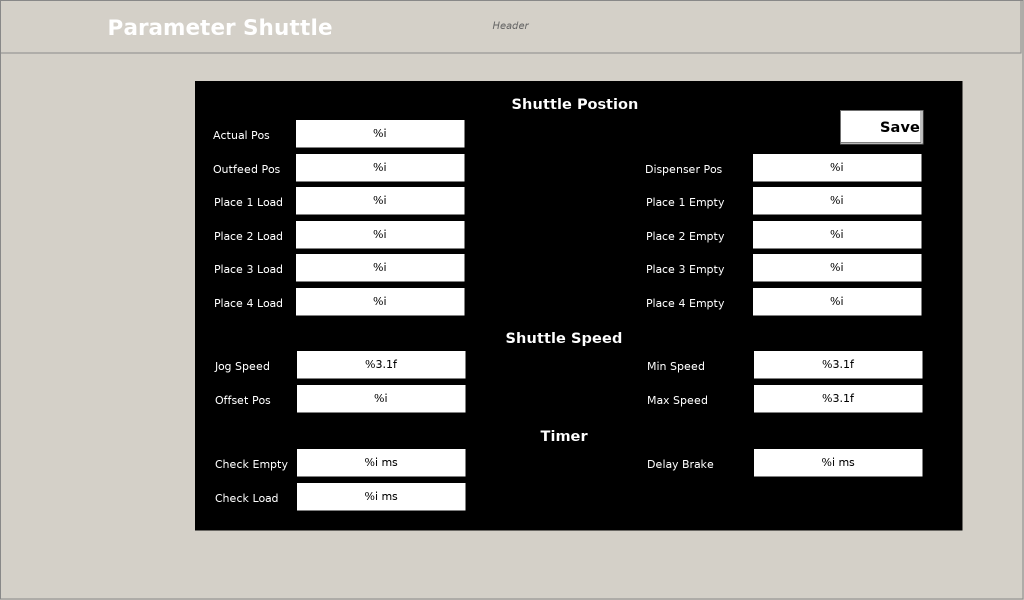
VISUALIZATION MShuttle  // 1024x600
    Frame (0,-2 1021x55)
        shows Header()
    Label (95,15 250x25), "Parameter Shuttle"
    RoundedRectangle (195,81 767x449)
    Label (223,84 704x40), "Shuttle Postion"
    Label (210,118 78x35), "Actual Pos"
    RoundedRectangle (295,119 170x29), "%i", text variable: InputOutput_GVL.ShuttlePosition
    Button (840,110 83x34), "Save", image: VisuSymbols.Symbols.Save
        tap InputOutput_GVL.TestMode[100]
    Label (210,152 78x35), "Outfeed Pos"
    RoundedRectangle (295,153 170x29), "%i", text variable: HMI_GVL.stShuttleSequence[0].PositionLoaded
        OnMouseClick: write the text variable via Default
    Label (642,152 102x35), "Dispenser Pos"
    RoundedRectangle (752,153 170x29), "%i", text variable: HMI_GVL.stShuttleSequence[0].PositionEmpty
        OnMouseClick: write the text variable via Default
    Label (211,185 78x35), "Place 1 Load"
    RoundedRectangle (295,186 170x29), "%i", text variable: HMI_GVL.stShuttleSequence[1].PositionLoaded
        OnMouseClick: write the text variable via Default
    Label (643,185 102x35), "Place 1 Empty"
    RoundedRectangle (752,186 170x29), "%i", text variable: HMI_GVL.stShuttleSequence[1].PositionEmpty
        OnMouseClick: write the text variable via Default
    Label (211,219 78x35), "Place 2 Load"
    RoundedRectangle (295,220 170x29), "%i", text variable: HMI_GVL.stShuttleSequence[2].PositionLoaded
        OnMouseClick: write the text variable via Default
    Label (643,219 102x35), "Place 2 Empty"
    RoundedRectangle (752,220 170x29), "%i", text variable: HMI_GVL.stShuttleSequence[2].PositionEmpty
        OnMouseClick: write the text variable via Default
    Label (211,252 78x35), "Place 3 Load"
    RoundedRectangle (295,253 170x29), "%i", text variable: HMI_GVL.stShuttleSequence[3].PositionLoaded
        OnMouseClick: write the text variable via Default
    Label (643,252 102x35), "Place 3 Empty"
    RoundedRectangle (752,253 170x29), "%i", text variable: HMI_GVL.stShuttleSequence[3].PositionEmpty
        OnMouseClick: write the text variable via Default
    Label (211,286 78x35), "Place 4 Load"
    RoundedRectangle (295,287 170x29), "%i", text variable: HMI_GVL.stShuttleSequence[4].PositionLoaded
        OnMouseClick: write the text variable via Default
    Label (643,286 102x35), "Place 4 Empty"
    RoundedRectangle (752,287 170x29), "%i", text variable: HMI_GVL.stShuttleSequence[4].PositionEmpty
        OnMouseClick: write the text variable via Default
    Label (212,318 704x40), "Shuttle Speed"
    Label (212,349 78x35), "Jog Speed"
    RoundedRectangle (296,350 170x29), "%3.1f", text variable: HMI_GVL.Shuttle_JogSpeed
        OnMouseClick: write the text variable via Default
    Label (644,349 102x35), "Min Speed"
    RoundedRectangle (753,350 170x29), "%3.1f", text variable: HMI_GVL.Shuttle_MinSpeed
        OnMouseClick: write the text variable via Default
    Label (212,383 78x35), "Offset Pos"
    RoundedRectangle (296,384 170x29), "%i", text variable: HMI_GVL.Shuttle_Offset
        OnMouseClick: write the text variable via Default
    Label (644,383 102x35), "Max Speed"
    RoundedRectangle (753,384 170x29), "%3.1f", text variable: HMI_GVL.Shuttle_MaxSpeed
        OnMouseClick: write the text variable via Default
    Label (212,416 704x40), "Timer"
    Label (212,447 78x35), "Check Empty"
    RoundedRectangle (296,448 170x29), "%i ms", text variable: HMI_GVL.Tmr_EmptyShuttle
        OnMouseClick: write the text variable via Default
    Label (644,447 102x35), "Delay Brake"
    RoundedRectangle (753,448 170x29), "%i ms", text variable: HMI_GVL.Tmr_BrakeShuttle
        OnMouseClick: write the text variable via Default
    Label (212,481 78x35), "Check Load"
    RoundedRectangle (296,482 170x29), "%i ms", text variable: HMI_GVL.Tmr_LoadedShuttle
        OnMouseClick: write the text variable via Default
END_VISUALIZATION

(* stored: Version 1.1.0.1, ProductVersion 3.1.4024.12
   Visu MShuttle: Id {5410681f-7c4a-472a-8e49-a5c1bcbc3460} *)
